// TIA Portal project "2022.06.13_PTO调试" (V17)

(* hardware
DEVICE "S7-1200 station_1"  S7-1200 Station
   slot 0: "Rack_0"  S7-1200 Rack  Rack  V1.0
   slot 1: "PLC_1"  CPU 1212C DC/DC/DC  6ES7 212-1AE40-0XB0  V4.5
   slot 2: "AI 4x13BIT/AQ 2x14BIT_1"  SM 1234 AI4/AQ2  6ES7 234-4HE30-0XB0  V1.0
*)

// ===== PLC "PLC_1"  CPU 1212C DC/DC/DC =====

VAR_GLOBAL   // PLC tag table "默认变量表"
   "液位测量" AT %IW96 : Word;
   "百分比" AT %MD40 : DWord;
   "模拟量输出通道" AT %MD44 : UDInt;
   "所需频率(1)" AT %MD0 : Real;
   "压力2模拟输入通道" AT %IW100 : Int;
   "液位" AT %MD4 : Real;
   "频率" AT %MD8 : Real;
   "Tag_2" AT %MD12 : Real;
   "模拟量输出" AT %QW96 : Int;
   "设定液位值" AT %MD20 : Real;
   "实际液位值" AT %MD24 : Real;
   "轴_1_脉冲" AT %Q0.0 : Bool;
   "轴_1_方向" AT %Q0.1 : Bool;
   "轴_1_LowHwLimitSwitch" AT %I0.0 : Bool;
   "轴_1_HighHwLimitSwitch" AT %I0.1 : Bool;
   "轴_1_PassiveHomingSwitch" AT %I0.2 : Bool;
   "轴_1_归位开关" AT %I0.3 : Bool;
END_VAR

DATA_BLOCK "轴_1"   // DB1, Motion_DB
{ S7_Optimized_Access := 'TRUE' }
AUTHOR : SIMATIC
FAMILY : BasicMC
NAME : TO_PosAx
VERSION : 8.0
// stored: InstanceOfName TO_PositioningAxis
"TO_PositioningAxis"
BEGIN
   // Axis.HomingReferencePointSwitch_AddressCU = %I0.3
   // Axis.LengthUnitNormalized.Distance = 1013
   // Axis.PositionLimitsMax_AddressCU = %I0.1
   // Axis.PositionLimitsMin_AddressCU = %I0.0
   // Axis.DirectionOutputEnabledCU = TRUE
   // Axis.OnlinePtoModeCU = 16#0000_0002
   // Axis.SelectedChannel2EnumCU = %Q0.1
   // Axis.SelectedChannel1EnumCU = %Q0.0
   // Pulse.MinDeltaDeltaFrequencyCU = 0.004
   // Pulse.MaxDeltaDeltaFrequencyCU = 1.0E+10
   // Pulse.MinDeltaFrequencyCU = 0.005
   // Pulse.MaxDeltaFrequencyCU = 9.5E+9
   // Pulse.MinFrequencyCU = 1.0
   // Pulse.MaxFrequencyCU = 100000.0
   // Pulse.OutputSourceCU = 16#0000_0000
   // Axis.SelectPTO = 0
END_DATA_BLOCK

ORGANIZATION_BLOCK "Main"   // OB1, LAD, ProgramCycle
TITLE = "Main Program Sweep (Cycle)"
{ S7_Optimized_Access := 'TRUE' }
VERSION : 0.1
   VAR_INPUT
      Initial_Call : Bool;   // Initial call of this OB
      Remanence : Bool;   // =True, if remanent data are available
   END_VAR
BEGIN
END_ORGANIZATION_BLOCK